{attribute 'OPC.UA.DA.StructuredType' := '1'}
FUNCTION_BLOCK FB_Sensor_GrowMedium_MOISTURE EXTENDS FB_BaseSensor IMPLEMENTS I_Device, I_Sensor

VAR
	
	bCAL: BOOL := FALSE;
	
	eSMState: (WAIT, CAL_DRY, CAL_WET, CALC_CORRECTION) := WAIT;

END_VAR
	
VAR PERSISTENT ;
	nMoisture_LOW_val: REAL;
	nMoisture_HIGH_val: REAL;
	
	nCurveGradient: REAL := 0.625; // 
	nCurveOffset: REAL := -2.5; // Defaults
END_VAR

calculate();
filter();

// Detect if any buttons in ignition have been pressed for Calibration
IF bCAL THEN 
	bCAL := FALSE;
	CASE eSMState OF
		WAIT:
			eSMState := CAL_DRY;
		CAL_DRY:
			eSMState := CAL_WET;
		CAL_WET:
			eSMState := CALC_CORRECTION;
	END_CASE
END_IF


CASE eSMState OF 
	WAIT:
		// wait here for a calibration command to be received
		eState := E_DeviceState.RUNNING;
	CAL_DRY:
		nMoisture_LOW_val 	:= nMeasuredCurrent;
		eState := E_DeviceState.CAL_STEP1;

	CAL_WET:
		nMoisture_HIGH_val 	:= nMeasuredCurrent;
		eState := E_DeviceState.CAL_STEP2;

	CALC_CORRECTION:
		nCurveGradient := 100.0 / (nMoisture_HIGH_val - nMoisture_LOW_val);
		nCurveOffset := 100.0 - (nCurveGradient * nMoisture_HIGH_val);
		eState := E_DeviceState.CAL_STEP3;
		eSMState := WAIT;
		
END_CASE

METHOD PRIVATE calculate : BOOL
VAR_INPUT
	
END_VAR
nMeasuredCurrent := (INT_TO_REAL(nRawInput)/GVL.nMaxADCOutput)*16.0 + 4.0; // in mA

// nCurrentValue := (nCurveGradient * nMeasuredCurrent) + nCurveOffset;

nCurrentValue := (nCurveGradient * nFilteredCurrent) + nCurveOffset; // delete this eventually
END_METHOD

METHOD calibrate : BOOL
VAR_INPUT
	
END_VAR

bCAL := TRUE;
END_METHOD

{warning 'add method implementation '}
METHOD disable : BOOL
bEnable := FALSE;
END_METHOD

{warning 'add method implementation '}
METHOD enable : BOOL
bEnable := TRUE;
END_METHOD

{warning 'add method implementation '}
METHOD FB_init : BOOL
VAR_INPUT
	(* if TRUE, the retain variables are initialized (warm start / cold start)*)
	bInitRetains	: BOOL;
	(* if TRUE, the instance afterwards gets moved into the copy code (online change)*)
	bInCopyCode	: BOOL;
	
	SensorID	: STRING(80);
	SensorDescr	: STRING(255);
	SensorType	: E_SensorType;
END_VAR
sID := SensorID;
sDescr := SensorDescr;
eSensorType := SensorType;
END_METHOD

{warning 'add method implementation '}
METHOD getType : E_SensorType
getType := eSensorType;
END_METHOD

{warning 'add method implementation '}
METHOD getValue : REAL
getValue := nCurrentValue;
END_METHOD

{warning 'add method implementation '}
METHOD write : BOOL
// use this method to initiated a hardware read from assigned IO if required
END_METHOD

END_FUNCTION_BLOCK

(* stored: Version 1.1.0.1, ProductVersion 3.1.4024.12
   POU FB_Sensor_GrowMedium_MOISTURE: Id {88957389-1c2c-4458-a94a-4cdf9eda6a51}, SpecialFunc None
   Method calculate: Id {be7a1123-9f60-4d09-9ba0-0ba768df3356}
   Method calibrate: Id {00ff78a3-5a41-48c6-b4f3-679db21971a2}
   Method disable: Id {6db9c88a-681b-4fc1-9e23-29f10af3ecd5}
   Method enable: Id {b42ee797-30b5-4118-86af-a4ab834733ad}
   Method FB_init: Id {b1e2a149-0ff5-4520-a291-2b94b5d27c2e}
   Method getType: Id {8288ddf3-20e2-438f-b80a-5e3e212915b9}
   Method getValue: Id {0431d3d5-5f7a-4a30-bb21-a4beac71f081}
   Method write: Id {b00fb345-eb3e-443d-97f4-cff1fe4eecd1} *)
